# EPICS autosave request: iocs/LambdaIOC/iocBoot/iocLambda/ADLambda_settings.req
$(P)$(R)HighEnergyThreshold
$(P)$(R)LowEnergyThreshold
